Fanuc KAREL source: compact_preamble.KL

PROGRAM KT00102
%NOLOCKGROUP
VAR
I1:INTEGER
Y2 : ARRAY[2] OF BYTE
OUT:REAL
BEGIN
I1=2
Y2[1]=3
OUT=((I1) / (Y2[1]))
END KT00102
